DATA_BLOCK "DB_StationSupervisor"
{ S7_Optimized_Access := 'TRUE' }
VERSION : 0.1
NON_RETAIN
"FB_StationSupervisor"
BEGIN
END_DATA_BLOCK
